PROGRAM FastPRG_1
VAR
	bolPlcStartupDone: BOOL := FALSE;
	bolHostInitDone: BOOL := FALSE;
	bolInitDone: BOOL := FALSE;
	strInstance: STRING;
	pCtrl_CIf: POINTER TO T_Ctrl_CIf;
	pTmpSIf_JUN: POINTER TO T_Ctrl_SIf_JUN;
	intState: INT;
	bolSetCmd: BOOL;
	jj: INT;
	bolCtrlRst: BOOL;
	/// Decision Point Heat Presses
	fbRFD_4: FB_RFR;
	fbJUN_4a: FB_JUN;
	fbJUN_4b: FB_JUN;
	fbJUN_5a: FB_JUN;
	fbJUN_5b: FB_JUN;
	fbJUN_6a: FB_JUN;
	fbJUN_6b: FB_JUN;
	/// Decision Point TLK
	fbRFD_15: FB_RFR;
	fbJUN_15a: FB_JUN;
	fbJUN_15b: FB_JUN;
	fbCHD_4: FB_CHD;
	pTmpSIf_CHD: POINTER TO T_Ctrl_SIf_CHD;
END_VAR

(*__________________________________________________________________________________________________
¦	
¦	Vistaprint Schweiz GmbH
¦	CH - 8401 Winterthur
¦
¦	www.vistaprint.ch - info@vistaprint.ch
¦___________________________________________________________________________________________________

Function desription:
call of all controller (FUB) for the fast task class.


History:
Version		Date			Author		Comment
---------------------------------------------------------------------------------------------------
0.00.1		16.09.2013		AVME/PRE	Start history
0.00.2		19.09.2013		AVME/PRE	Implement new Base Concept
0.00.3		08.10.2013		VP/RE		Optimizations FAT Bürglistrasse version
0.00.4		24.10.2013		AVME/MRU	CHD added, New BASE_PLC 0.3.3.0
0.00.5		18.11.2013		AVME/MRU	CHD Parameter changed
0.00.6		30.01.2013		VP/RE		JUN parameter changed
___________________________________________________________________________________________________*)

// -----------------------------------------------------------------------------------------------
// Initialize the PLC Parameter and check the PLC health
// -----------------------------------------------------------------------------------------------
IF (NOT bolPlcStartupDone) THEN
	bolPlcStartupDone := TRUE;	
	
	// init	
	// Decision Point Heat Presses
	g_a_pFunRFD[1] := ADR(fbRFD_4);

	fbJUN_4a.iniAllCtrlArrays(ADR(g_a_pCtrlInst),ADR(g_a_pCtrlCIf),E_CtrlId.JUN_4a);                   // init and entry fb_instance in global fb pointer array
	pTmpSIf_JUN := fbJUN_4a.getCtrlSIf();
	pTmpSIf_JUN^.Cfg.dinTargetNr := 1;	
	pTmpSIf_JUN^.Par.udiOpenTime_ms:= 20;
	pTmpSIf_JUN^.Par.udiCloseTime_ms:= 10;
	pTmpSIf_JUN^.Par.udiPassTime_ms:= 4000;
	pTmpSIf_JUN^.Par.dinOpenWay_um:= 200000;
	pTmpSIf_JUN^.Par.dinPosition_um := 2340000;
	
	fbJUN_4b.iniAllCtrlArrays(ADR(g_a_pCtrlInst),ADR(g_a_pCtrlCIf),E_CtrlId.JUN_4b);                  // init and entry fb_instance in global fb pointer array
	pTmpSIf_JUN := fbJUN_4b.getCtrlSIf();
	pTmpSIf_JUN^.Cfg.dinTargetNr := 2;	
	pTmpSIf_JUN^.Par.udiOpenTime_ms:= 20;
	pTmpSIf_JUN^.Par.udiCloseTime_ms:= 10;
	pTmpSIf_JUN^.Par.udiPassTime_ms:= 4000;
	pTmpSIf_JUN^.Par.dinOpenWay_um:= 200000;
	pTmpSIf_JUN^.Par.dinPosition_um := 3055000;

	fbJUN_5a.iniAllCtrlArrays(ADR(g_a_pCtrlInst),ADR(g_a_pCtrlCIf),E_CtrlId.JUN_5a);                   // init and entry fb_instance in global fb pointer array
	pTmpSIf_JUN := fbJUN_5a.getCtrlSIf();
	pTmpSIf_JUN^.Cfg.dinTargetNr := 1;	
	pTmpSIf_JUN^.Par.udiOpenTime_ms:= 20;
	pTmpSIf_JUN^.Par.udiCloseTime_ms:= 10;
	pTmpSIf_JUN^.Par.udiPassTime_ms:= 4000;
	pTmpSIf_JUN^.Par.dinOpenWay_um:= 200000;
	pTmpSIf_JUN^.Par.dinPosition_um := 2340000;
	
	fbJUN_5b.iniAllCtrlArrays(ADR(g_a_pCtrlInst),ADR(g_a_pCtrlCIf),E_CtrlId.JUN_5b);                  // init and entry fb_instance in global fb pointer array
	pTmpSIf_JUN := fbJUN_5b.getCtrlSIf();
	pTmpSIf_JUN^.Cfg.dinTargetNr := 2;	
	pTmpSIf_JUN^.Par.udiOpenTime_ms:= 20;
	pTmpSIf_JUN^.Par.udiCloseTime_ms:= 10;
	pTmpSIf_JUN^.Par.udiPassTime_ms:= 4000;
	pTmpSIf_JUN^.Par.dinOpenWay_um:= 200000;
	pTmpSIf_JUN^.Par.dinPosition_um := 3055000;
	
	fbJUN_6a.iniAllCtrlArrays(ADR(g_a_pCtrlInst),ADR(g_a_pCtrlCIf),E_CtrlId.JUN_6a);                   // init and entry fb_instance in global fb pointer array
	pTmpSIf_JUN := fbJUN_6a.getCtrlSIf();
	pTmpSIf_JUN^.Cfg.dinTargetNr := 1;	
	pTmpSIf_JUN^.Par.udiOpenTime_ms:= 20;
	pTmpSIf_JUN^.Par.udiCloseTime_ms:= 10;
	pTmpSIf_JUN^.Par.udiPassTime_ms:= 4000;
	pTmpSIf_JUN^.Par.dinOpenWay_um:= 200000;
	pTmpSIf_JUN^.Par.dinPosition_um := 2340000;
	
	fbJUN_6b.iniAllCtrlArrays(ADR(g_a_pCtrlInst),ADR(g_a_pCtrlCIf),E_CtrlId.JUN_6b);                  // init and entry fb_instance in global fb pointer array
	pTmpSIf_JUN := fbJUN_6b.getCtrlSIf();
	pTmpSIf_JUN^.Cfg.dinTargetNr := 2;	
	pTmpSIf_JUN^.Par.udiOpenTime_ms:= 20;
	pTmpSIf_JUN^.Par.udiCloseTime_ms:= 10;
	pTmpSIf_JUN^.Par.udiPassTime_ms:= 4000;
	pTmpSIf_JUN^.Par.dinOpenWay_um:= 200000;
	pTmpSIf_JUN^.Par.dinPosition_um := 3055000;
	
	// Decision Point TLK
	g_a_pFunRFD[2] := ADR(fbRFD_15);

	fbJUN_15a.iniAllCtrlArrays(ADR(g_a_pCtrlInst),ADR(g_a_pCtrlCIf),E_CtrlId.JUN_15a);  // init and entry fb_instance in global fb pointer array
	pTmpSIf_JUN := fbJUN_15a.getCtrlSIf();
	pTmpSIf_JUN^.Cfg.dinTargetNr := 1;
	pTmpSIf_JUN^.Par.udiOpenTime_ms:= 20;
	pTmpSIf_JUN^.Par.udiCloseTime_ms:= 10;
	pTmpSIf_JUN^.Par.udiPassTime_ms:= 4000;
	pTmpSIf_JUN^.Par.dinOpenWay_um:= 350000;
	pTmpSIf_JUN^.Par.dinPosition_um := 6140000;
	

	fbJUN_15b.iniAllCtrlArrays(ADR(g_a_pCtrlInst),ADR(g_a_pCtrlCIf),E_CtrlId.JUN_15b); // init and entry fb_instance in global fb pointer array
	pTmpSIf_JUN := fbJUN_15b.getCtrlSIf();
	pTmpSIf_JUN^.Cfg.dinTargetNr := 2;	
	pTmpSIf_JUN^.Par.udiOpenTime_ms:= 20;
	pTmpSIf_JUN^.Par.udiCloseTime_ms:= 10;
	pTmpSIf_JUN^.Par.udiPassTime_ms:= 4000;
	pTmpSIf_JUN^.Par.dinOpenWay_um:= 350000;
	pTmpSIf_JUN^.Par.dinPosition_um := 7240000;
	
	// ----------
	// CHD_4
	// ----------	
	fbCHD_4.iniAllCtrlArrays(ADR(g_a_pCtrlInst),ADR(g_a_pCtrlCIf),E_CtrlId.CHD_4);     	// init and entry fb_instance in global fb pointer array
	pTmpSIf_CHD := fbCHD_4.getCtrlSIf();
	// CHD_4 - configuration
	pTmpSIf_CHD^.Cfg.bolHasInconsistentHangerSensor := FALSE;
	pTmpSIf_CHD^.Cfg.bolHasEmptyHangerSensor := TRUE;
	pTmpSIf_CHD^.Cfg.bolStopAtRejact := FALSE;
	// CHD_4 - parameter
	pTmpSIf_CHD^.Par.dinPosition_um := 190000-110000; // Position - open befor there // 200000;
	pTmpSIf_CHD^.Par.dinOpenWay_um := 200000; // 200000;
	pTmpSIf_CHD^.Par.dinDistanceBetweenSensors_um := 200000; // not used, only 1 Sensor
	pTmpSIf_CHD^.Par.dinPinDistance_um := 305000;
	pTmpSIf_CHD^.Par.udinTimeUntilJam_ms := 1000;
	pTmpSIf_CHD^.Par.udiPulseLengthBlowValve_ms := 200;
	pTmpSIf_CHD^.Par.udiIntervalLengthBlowValve_ms := 60000;

	g_uinStartProzess:=1; // For StartUp order

END_IF
// -----------------------------------------------------------------------------------------------


// -----------------------------------------------------------------------------------------------
// The host system is downloading all parameter at startup. 
// bolPlcStartupDone will be set to true after the Host is done with the initialization
// -----------------------------------------------------------------------------------------------
IF (bolPlcStartupDone AND (NOT bolHostInitDone) AND (NOT bolInitDone) AND (g_uinStartProzess>=c_uinCntTaskClass)) THEN
	bolHostInitDone := TRUE;
	g_uinStartProzess := 11; // For StartUp order
END_IF
// -----------------------------------------------------------------------------------------------


// -----------------------------------------------------------------------------------------------
// Start PLC code initialization
// -----------------------------------------------------------------------------------------------
IF (NOT bolInitDone AND bolPlcStartupDone AND bolHostInitDone AND (g_uinStartProzess>=(10+c_uinCntTaskClass))) THEN
	g_uinStartProzess := 21; // For StartUp order
	bolInitDone := TRUE;
END_IF
// -----------------------------------------------------------------------------------------------

// -----------------------------------------------------------------------------------------------
// Normal Run mode after all the initialization is done
// -----------------------------------------------------------------------------------------------
IF (bolInitDone AND bolPlcStartupDone AND bolHostInitDone AND (g_uinStartProzess>=(20+c_uinCntTaskClass))) THEN
	
	//****************************************************************************************************
	// cyclic controller calls
	//****************************************************************************************************
	// Decision Point Heat Presses
	fbRFD_4();
	fbJUN_4a.In_bolPassed := In_4_0_B12_Hanger_Acknowledged;
	fbJUN_4a();
	Out_4_0_Y11_Junction := fbJUN_4a.Out_bolOpen;
	
	fbJUN_4b.In_bolPassed := In_4_0_B15_Hanger_Acknowledged;
	fbJUN_4b();
	Out_4_0_Y14_Junction := fbJUN_4b.Out_bolOpen;

	fbJUN_5a.In_bolPassed := In_4_0_B22_Hanger_Acknowledged;
	fbJUN_5a();
	Out_4_0_Y21_Junction := fbJUN_5a.Out_bolOpen;
	
	fbJUN_5b.In_bolPassed := In_4_0_B24_Hanger_Acknowledged;
	fbJUN_5b();
	Out_4_0_Y23_Junction := fbJUN_5b.Out_bolOpen;
	
	fbJUN_6a.In_bolPassed := In_4_0_B26_Hanger_Acknowledged;
	fbJUN_6a();
	Out_4_0_Y25_Junction := fbJUN_6a.Out_bolOpen;
	
	fbJUN_6b.In_bolPassed := In_4_0_B28_Hanger_Acknowledged;
	fbJUN_6b();
	Out_4_0_Y27_Junction := fbJUN_6b.Out_bolOpen;
	
	// Decision Point TLK
	fbRFD_15();
	fbJUN_15a.In_bolPassed := In_15_0_B15a_Dischare_Acknowledged;
	fbJUN_15a();
	Out_15_Y3_Junction := fbJUN_15a.Out_bolOpen;
	
	fbJUN_15b.In_bolPassed := In_15_0_B17a_Dischare_Acknowledged;
	fbJUN_15b();
	Out_15_Y4_Junction := fbJUN_15b.Out_bolOpen;

	// Inputs
	fbCHD_4.In_bolDoubleHanger := In_4_0_B4_Crossed_Hanger_Detection;
	fbCHD_4.In_bolPassed := In_4_0_B16_Rail_Full;
	fbCHD_4.In_bolEmptyHanger := In_4_0_B3_Empty_Hanger_Detection;
	// Function call
	fbCHD_4();
	// Outputs
	Out_4_0_Y6_Junction := fbCHD_4.Out_bolOpen;
	Out_4_0_Y5_Blowing_Light_Barrier := fbCHD_4.Out_bolBlow;

END_IF
// -----------------------------------------------------------------------------------------------

END_PROGRAM

(* stored: Version 1.1.0.1, ProductVersion 3.1.0.23
   POU FastPRG_1: Id {b624d175-54f8-4f4a-ae3e-53272a249758} *)
